(* CODESYS project WagoAppCloud_Influxdb_1.8.ecp
   Company: WAGO
   Title: WagoAppCloud_CostumerProtocol
   Description: Example for the Cloud Conectivity using MQTT with the own customer data strucure
   Author: wago / u014791
   Version: 1.0.0.0

Project tree, tasks and I/O mapping:
  Edge : Edge Controller PIO3, WAGO, order no. 0752-8303, version 5.15.4.20
    application Application
      libraries: WagoAppString, 1.6.3.1 (WAGO); WagoAppCloud, * (WAGO); Util, * (System); WagoAppTime, 1.7.3.3 (WAGO)
      task Task (cyclic, interval t#10ms, priority 14) calls PLC_PRG
      program Status_NativeMQTT [ST]
      program Publish_NativeMQTT [ST]
      program PLC_PRG [ST]
    ProjectConfiguration
    ProjectConfigurationTxt
    CANbus
    MODBUS
      MODBUS : MODBUS, WAGO, order no. n/a, version 1.1.1.15
    Serial
      COM1 : COM1, WAGO, version 0.0.0.19
    TP600_Onboard_IO : TP600 Onboard IO, WAGO, version 0.0.1.2
        unmapped channels: _IN, _OUT
    Common.PCI
  TP600 : TP600 10.1 1280x800 PIO3 CP , WAGO, order no. 0762-5304, version 5.15.4.20
    application Application
      libraries: WagoAppString, 1.6.3.1 (WAGO); WagoAppCloud, * (WAGO); Util, * (System); WagoAppTime, 1.7.3.3 (WAGO)
      task Task (cyclic, interval t#10ms, priority 14) calls PLC_PRG
      program Status_NativeMQTT [ST]
      program Publish_NativeMQTT [ST]
      program PLC_PRG [ST]
    ProjectConfigurationTxt
    ProjectConfiguration
    MODBUS
      MODBUS : MODBUS, WAGO, order no. n/a, version 1.1.1.15
    CANbus
    TP600_Onboard_IO : TP600 Onboard IO, WAGO, version 0.0.1.2
        unmapped channels: _IN, _OUT
    Common.PCI
    Serial
      COM1 : COM1, WAGO, version 0.0.0.19
  00000000-0000-0000-0000-000000000000|C:\Users\u042194\AppData\Local\Temp\0a333301e76e4166a24b2b16dca87435\ProjectCfg.txt
  00000000-0000-0000-0000-000000000000|C:\Users\u042194\AppData\Local\Temp\cacff6e159c24479a4cea757bd311a24\Project.xml
  00000000-0000-0000-0000-000000000000|C:\Users\u042194\AppData\Local\Temp\5feddc19d5d94271be77a83e116637d0\Project.xml
  00000000-0000-0000-0000-000000000000|C:\Users\u042194\AppData\Local\Temp\0871f40602084dc4a0da722e5aa72ddc\ProjectCfg.txt
*)

// Edge/Application/PLC_PRG
PROGRAM PLC_PRG
VAR
END_VAR

Publish_NativeMQTT();	
Status_NativeMQTT();

END_PROGRAM

// Edge/Application/Publish_NativeMQTT
// !!! IMPORTANT !!!
// Some cloud platforms have limitations on their MQTT-Implementation.
// Typically the supported payload size is significantly less then told by MQTT-Specification:
// it is 128KB for IBM Bluemix and Amazon Web Services (https://docs.aws.amazon.com/iot/latest/developerguide/protocols.html)
// Other known limitations are related to Quality Of Service Level, Retain message flag, ...
// !!! IMPORTANT !!!

// Purpose of the example program: Primitive JSON document shall periodically be published via dataagent daemon

PROGRAM Publish_NativeMQTT
VAR
	MyInterval		: TIME := T#1S;
	Timer			: TON;
	
	dwMyCounter 	: DWORD := 1;
	MyString 		: STRING(255);
	aBuffer			: ARRAY[0..255] OF BYTE;
	dwBytesCount 	: DWORD;
	
	oFbPublish 		: WagoAppCloud.FbPublishMQTT;
	xMyTrigger		: BOOL := FALSE;
	dwBusyCounter	: DWORD := 0;
	dwErrorCounter	: DWORD := 0;
	signal: INT;
	oGen: Util.GEN;
END_VAR

dwMyCounter := dwMyCounter + 1;

Timer(IN := TRUE, PT := MyInterval);
IF Timer.Q THEN
	Timer(IN := FALSE);

	IF NOT oFbPublish.xBusy THEN
		// Write primitive JSON into string (use WagoAppJson library for advanced JSON functionalities)
		//MyString := CONCAT('{"Value":', DWORD_TO_STRING(dwMyCounter));
			//MyString := CONCAT(MyString,'}');
			
			MyString:=CONCAT4('processdata,source=Edge counter=',TO_STRING(dwMyCounter), ',signal=', TO_STRING(signal));//, ' ', TO_STRING(TO_LWORD(WagoAppTime.FuGetLongTime())));
		
		//MyString := DWORD_TO_STRING(dwMyCounter);
		// Copy JSON to buffer
		dwBytesCount := Length(MyString);
		MemCopy(pDest := ADR(aBuffer), pSource := ADR(MyString), udiSize := dwBytesCount);
		// Trigger the transmission
		xMyTrigger := TRUE;
	ELSE
		// Busy statistics counter
		dwBusyCounter := dwBusyCounter + 1;
	END_IF
	
	IF oFbPublish.xError THEN
		// Error statistics counter
		dwErrorCounter := dwErrorCounter + 1;
	END_IF
	
END_IF


oGen(
	MODE:=COSINUS , 
	BASE:=TRUE , 
	PERIOD:=T#1M , 
	CYCLES:= , 
	AMPLITUDE:=100 , 
	RESET:= , 
	OUT=>signal );

// Trigger MQTT publish
oFbPublish(sTopic := 'wago/subtopic',
			eQualityOfService := 1,
			dwSize := dwBytesCount,
			aData := aBuffer,
			xTrigger := xMyTrigger);

END_PROGRAM

// TP600/Application/Publish_NativeMQTT
// !!! IMPORTANT !!!
// Some cloud platforms have limitations on their MQTT-Implementation.
// Typically the supported payload size is significantly less then told by MQTT-Specification:
// it is 128KB for IBM Bluemix and Amazon Web Services (https://docs.aws.amazon.com/iot/latest/developerguide/protocols.html)
// Other known limitations are related to Quality Of Service Level, Retain message flag, ...
// !!! IMPORTANT !!!

// Purpose of the example program: Primitive JSON document shall periodically be published via dataagent daemon

PROGRAM Publish_NativeMQTT
VAR
	MyInterval		: TIME := T#1S;
	Timer			: TON;
	
	dwMyCounter 	: DWORD := 1;
	MyString 		: STRING(255);
	aBuffer			: ARRAY[0..255] OF BYTE;
	dwBytesCount 	: DWORD;
	
	oFbPublish 		: WagoAppCloud.FbPublishMQTT;
	xMyTrigger		: BOOL := FALSE;
	dwBusyCounter	: DWORD := 0;
	dwErrorCounter	: DWORD := 0;
	signal: INT;
	oGen: Util.GEN;
END_VAR

dwMyCounter := dwMyCounter + 1;

Timer(IN := TRUE, PT := MyInterval);
IF Timer.Q THEN
	Timer(IN := FALSE);

	IF NOT oFbPublish.xBusy THEN
		// Write primitive JSON into string (use WagoAppJson library for advanced JSON functionalities)
		//MyString := CONCAT('{"Value":', DWORD_TO_STRING(dwMyCounter));
			//MyString := CONCAT(MyString,'}');
			
			MyString:=CONCAT4('processdata,source=TP600 counter=',TO_STRING(dwMyCounter), ',signal=', TO_STRING(signal));//, ' ', TO_STRING(TO_LWORD(WagoAppTime.FuGetLongTime())));
		
		//MyString := DWORD_TO_STRING(dwMyCounter);
		// Copy JSON to buffer
		dwBytesCount := Length(MyString);
		MemCopy(pDest := ADR(aBuffer), pSource := ADR(MyString), udiSize := dwBytesCount);
		// Trigger the transmission
		xMyTrigger := TRUE;
	ELSE
		// Busy statistics counter
		dwBusyCounter := dwBusyCounter + 1;
	END_IF
	
	IF oFbPublish.xError THEN
		// Error statistics counter
		dwErrorCounter := dwErrorCounter + 1;
	END_IF
	
END_IF


oGen(
	MODE:=COSINUS , 
	BASE:=TRUE , 
	PERIOD:=T#1M , 
	CYCLES:= , 
	AMPLITUDE:=100 , 
	RESET:= , 
	OUT=>signal );

// Trigger MQTT publish
oFbPublish(sTopic := 'wago/subtopic',
			eQualityOfService := 1,
			dwSize := dwBytesCount,
			aData := aBuffer,
			xTrigger := xMyTrigger);

END_PROGRAM

// Edge/Application/Status_NativeMQTT
// Purpose of the example program: Check status of Native MQTT
PROGRAM Status_NativeMQTT
VAR
	oFbStatus 			: WagoAppCloud.FbStatus_NativeMQTT;
	xMyError			: BOOL := FALSE;
	xConnectedToMyCloud	: BOOL := FALSE;
	rMyFillLevel		: REAL := 0;
	uliMyOutgoingBlocks	: ULINT := 0;
END_VAR

// Will detect new values every 5 seconds
oFbStatus(xEnabled := TRUE,
		   xError => xMyError,
		   xCloudConnected => xConnectedToMyCloud,			// Will be FALSE after network timeout occured 
		   rCacheFillLevel => rMyFillLevel,					// Increasing value indicates bad network or overload
		   uliOutgoingDataBlocks => uliMyOutgoingBlocks);  	// Only for QoS 1 and 2. Increasing value indicates bad network or overload

END_PROGRAM

// TP600/Application/Status_NativeMQTT
// Purpose of the example program: Check status of Native MQTT
PROGRAM Status_NativeMQTT
VAR
	oFbStatus 			: WagoAppCloud.FbStatus_NativeMQTT;
	xMyError			: BOOL := FALSE;
	xConnectedToMyCloud	: BOOL := FALSE;
	rMyFillLevel		: REAL := 0;
	uliMyOutgoingBlocks	: ULINT := 0;
END_VAR

// Will detect new values every 5 seconds
oFbStatus(xEnabled := TRUE,
		   xError => xMyError,
		   xCloudConnected => xConnectedToMyCloud,			// Will be FALSE after network timeout occured 
		   rCacheFillLevel => rMyFillLevel,					// Increasing value indicates bad network or overload
		   uliOutgoingDataBlocks => uliMyOutgoingBlocks);  	// Only for QoS 1 and 2. Increasing value indicates bad network or overload

END_PROGRAM

// TP600/Application/PLC_PRG
PROGRAM PLC_PRG
VAR
END_VAR

Publish_NativeMQTT();	
Status_NativeMQTT();

END_PROGRAM
